{attribute 'GeneratedUsingTerminal: EL2595-0000-0018'}
{attribute addProperty BoxType "EL2595-0000-0018"}
{attribute addProperty Id "StatusAT %I*Status_3BF44A816"}
{attribute addProperty CRC "2933432618"}
{attribute addProperty Size "6"}
TYPE DOX_Status_AED8A12A :
STRUCT
	{attribute addProperty Name "Status"}
	Status AT %I* : Status_3BF44A81;
END_STRUCT
END_TYPE

(* stored: Version 1.2.0.0, ProductVersion 3.1.4024.9
   DUT DOX_Status_AED8A12A: Id {e1cd85f2-fa44-479e-b90b-e217d996115c} *)
